# EPICS IOC start-up script: iocsh/LakeShore_340.iocsh
# ### LakeShore_340.iocsh ###

#- ###################################################
#- PREFIX         - IOC Prefix
#- INSTANCE       - Instance Prefix
#- PORT           - Serial port name
#- IP             - Location of IP module
#- ###################################################

iocshLoad("$(IP)/iocsh/setSerialParams.iocsh", "BAUD=9600, BITS=8, STOP=1, PARITY=none")

asynOctetSetInputEos( "$(PORT)", -1, "\r")
asynOctetSetOutputEos("$(PORT)", -1, "\r")

dbLoadRecords("$(IP)/ipApp/Db/LakeShore340.db", "P=$(PREFIX),Q=$(INSTANCE),PORT=$(PORT)")
